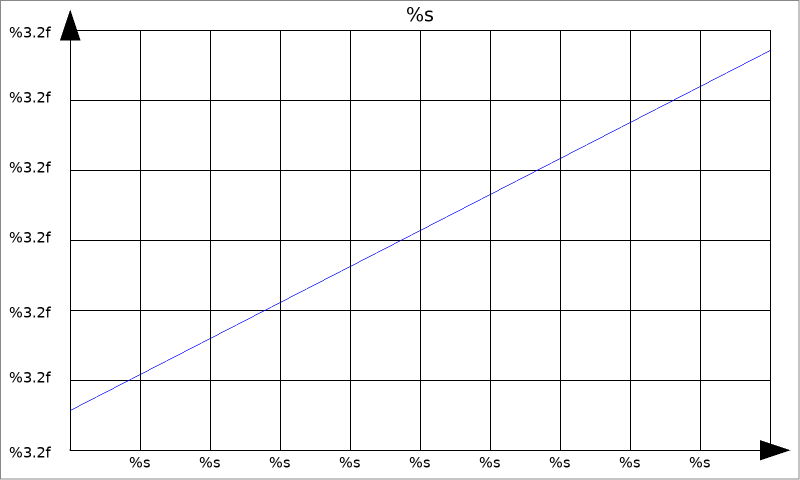
VISUALIZATION Trend_800_480  // 800x480
VAR_INPUT
	Header : WSTRING;
END_VAR
VAR_IN_OUT
	fb_TrendChanel1: FB_TrandChanel;
END_VAR
    Polyline (70,20) (70,450) (770,450)
    Polygon (70,10) (80,40) (60,40)
    Polygon (790,450) (760,460) (760,440)
    Line (70,380) (770,380)
    Line (70,310) (770,310)
    Line (70,240) (770,240)
    Line (70,170) (770,170)
    Line (70,100) (770,100)
    Polyline (70,410) (770,50)
    Rectangle (0,440 60x25), "%3.2f", text variable: fb_TrendChanel1.X_AxisNames[1]
    Rectangle (0,365 60x25), "%3.2f", text variable: fb_TrendChanel1.X_AxisNames[2]
    Rectangle (0,300 60x25), "%3.2f", text variable: fb_TrendChanel1.X_AxisNames[3]
    Rectangle (0,225 60x25), "%3.2f", text variable: fb_TrendChanel1.X_AxisNames[4]
    Rectangle (0,155 60x25), "%3.2f", text variable: fb_TrendChanel1.X_AxisNames[5]
    Rectangle (0,85 60x25), "%3.2f", text variable: fb_TrendChanel1.X_AxisNames[6]
    Rectangle (0,20 60x25), "%3.2f", text variable: fb_TrendChanel1.X_AxisNames[7]
    Rectangle (105,450 70x25), "%s", text variable: fb_TrendChanel1.Y_AxisNames[1]
    Rectangle (175,450 70x25), "%s", text variable: fb_TrendChanel1.Y_AxisNames[2]
    Rectangle (245,450 70x25), "%s", text variable: fb_TrendChanel1.Y_AxisNames[3]
    Rectangle (315,450 70x25), "%s", text variable: fb_TrendChanel1.Y_AxisNames[4]
    Rectangle (385,450 70x25), "%s", text variable: fb_TrendChanel1.Y_AxisNames[5]
    Rectangle (455,450 70x25), "%s", text variable: fb_TrendChanel1.Y_AxisNames[6]
    Rectangle (525,450 70x25), "%s", text variable: fb_TrendChanel1.Y_AxisNames[7]
    Rectangle (595,450 70x25), "%s", text variable: fb_TrendChanel1.Y_AxisNames[8]
    Rectangle (665,450 70x25), "%s", text variable: fb_TrendChanel1.Y_AxisNames[9]
    Rectangle (210,0 420x30), "%s", text variable: Header
    Line (70,30) (770,30)
    Line (140,30) (140,450)
    Line (210,30) (210,450)
    Line (280,30) (280,450)
    Line (350,30) (350,450)
    Line (420,30) (420,450)
    Line (490,30) (490,450)
    Line (560,30) (560,450)
    Line (630,30) (630,450)
    Line (700,30) (700,450)
    Line (770,30) (770,450)
END_VISUALIZATION

(* stored: Version 1.1.0.1, ProductVersion 3.1.4024.2
   Visu Trend_800_480: Id {c7f9bdbc-a7d4-4a18-b949-a6bd287acaf6} *)
